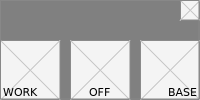
VISUALIZATION VisuCylinderHorLeftCtrl  // 200x100
VAR_IN_OUT
	fbVisuCylinder: FB_VISU_CYLINDER;
END_VAR
    Rectangle (0,0 200x100)
    Image (140,40 60x60), "BASE", image: VisuSymbols.Symbols.TriangleRight
        OnMouseClick: execute {
            fbVisuCylinder.bMoveToBase:=TRUE;
            fbVisuCylinder.bMoveToWork:=FALSE;
            fbVisuCylinder.bAllOff:=false;
            fbVisuCylinder.bFrameInvisible:= true;
        }
    Image (0,40 60x60), "WORK", image: VisuSymbols.Symbols.TriangleLeft
        OnMouseClick: execute {
            fbVisuCylinder.bMoveToWork:=TRUE;
            fbVisuCylinder.bMoveToBase:=FALSE;
            fbVisuCylinder.bAllOff:=false;
            fbVisuCylinder.bFrameInvisible:= true;
        }
    Image (180,0 20x20), image: VisuSymbols.Symbols.Wrong
        OnMouseDown: execute { fbVisuCylinder.bFrameInvisible:= true; }
    Image (70,40 60x60), "OFF", image: VisuSymbols.Symbols.Stop
        OnMouseClick: execute {
            fbVisuCylinder.bMoveToBase:=FALSE;
            fbVisuCylinder.bMoveToWork:=FALSE;
            fbVisuCylinder.bAllOff:=TRUE;
            fbVisuCylinder.bFrameInvisible:= true;
        }
END_VISUALIZATION

(* stored: Version 1.1.0.1, ProductVersion 3.1.4024.12
   Visu VisuCylinderHorLeftCtrl: Id {e818f303-3d2f-4818-8f22-45a40085a465} *)
